RESOURCE_TYPE TEST_RES (* Empty resource type for mapping tests *)
  (* Standard: 61499-1 *)
  (* Version 1.0, 2026-02-23, test, 4diac tests *)
END_RESOURCE_TYPE
